FUNCTION_BLOCK FB_SimpleNciSequence
VAR_INPUT
	bExecute			: BOOL;
END_VAR
VAR_OUTPUT
	bBusy				: BOOL;
	bError				: BOOL;
	bDone				: BOOL;
END_VAR
VAR_IN_OUT
	stX					: AXIS_REF;
	stY					: AXIS_REF;
	stZ					: AXIS_REF;
	stQ1				: AXIS_REF;
	stQ2				: AXIS_REF;
	stQ3				: AXIS_REF;
	stItpToPlc			: NCTOPLC_NCICHANNEL_REF;
	stPlcToItp			: PLCTONC_NCICHANNEL_REF;
END_VAR
VAR
	nState				: UDINT	:= 0;
	nErrorState			: UDINT;
	
	fbBuildGroup		: CfgBuildExt3DGroup;
	fbLoadGCode			: ItpLoadProgEx;
	fbStartGCode		: ItpStartStopEx;
	fbClearGroup		: CfgReconfigGroup;
	fbConfirmHsk		: ItpConfirmHsk;
	
	nInterpreterState	: UDINT	:= 0;
	bConfirmHsk			: BOOL	:= FALSE;
	
//	sPrgName			: STRING(255) := 'GST_SampleFunctions.nc'; //'first.nc';
//	sPrgName			: STRING(255) := 'first.nc'; //'';
//	sPrgName			: STRING(255) := 'sample.nc'; //'';
	sPrgName			: STRING(255) := 'functionsExample.nc'; //'';
	
	
END_VAR

CASE nState OF
0:
	IF bExecute THEN
		bBusy	:= TRUE;
		bDone	:= FALSE;
		bError	:= FALSE;
		nErrorState	:= nState;
		nState	:= 10;
	END_IF	
	
10:
	// first build interpolation group 
	nInterpreterState	:= ItpGetStateInterpreter(sNciToPlc:=stItpToPlc);
	IF nInterpreterState = Tc2_NCI.NCI_INTERPRETER_IDLE THEN
		fbBuildGroup(
			bExecute	:= TRUE, 
			nGroupId	:= ItpGetGroupId(sNciToPlc:=stItpToPlc) , 
			nXAxisId	:= stX.NcToPlc.AxisId, 
			nYAxisId	:= stY.NcToPlc.AxisId, 
			nZAxisId	:= stZ.NcToPlc.AxisId, 
			nQ1AxisId	:= stQ1.NcToPlc.AxisId, 
			nQ2AxisId	:= stQ2.NcToPlc.AxisId, 
			nQ3AxisId	:= stQ3.NcToPlc.AxisId, 
			nQ4AxisId	:= 0, 
			nQ5AxisId	:= 0, 
			tTimeOut	:= , 
			bBusy		=> , 
			bErr		=> , 
			nErrId		=> );
			
		IF NOT fbBuildGroup.bBusy THEN
			IF NOT fbBuildGroup.bErr THEN
				nState	:= 20;
			ELSE
				(* add error handling *)
				nErrorState	:= nState;
				bBusy	:= FALSE;
				bError	:= TRUE;
				nState	:= 9999;
			END_IF
			fbBuildGroup(bExecute:=FALSE); 
		END_IF
	END_IF
	
20:
	// load g-code file 
	// pls. ensure that first.nc is available in TwinCAT\MC\NCI-folder 
	fbLoadGCode(
		sNciToPlc	:= stItpToPlc, 
		bExecute	:= TRUE, 
		sPrg		:= sPrgName, 
		nLength		:= INT_TO_UDINT(LEN(sPrgName)), 
		tTimeOut	:= , 
		bBusy		=> , 
		bErr		=> , 
		nErrId		=> );
		
	IF NOT fbLoadGCode.bBusy THEN
		IF NOT fbLoadGCode.bErr THEN
			nState	:= 30;
		ELSE
			(* add error handling *)
			nErrorState	:= nState;
			bBusy	:= FALSE;
			bError	:= TRUE;
			nState	:= 9999;				
		END_IF
		fbLoadGCode(sNciToPlc:=stItpToPlc, bExecute:=FALSE); 
	END_IF
	
30:
	// we have to check the status of the interpreter. It has to be in ready state, in case of loading the program successfully.
	nInterpreterState	:= ItpGetStateInterpreter(sNciToPlc:=stItpToPlc);
	IF nInterpreterState = Tc2_NCI.NCI_INTERPRETER_READY THEN
		nState	:= 40;
	ELSE
		(* add error handling *)
		nErrorState	:= nState;
		bBusy	:= FALSE;
		bError	:= TRUE;
		nState	:= 9999;				
	END_IF
	
40:
	// start g-code file
	fbStartGCode(
		bStart		:=TRUE, 
		bStop		:=FALSE, 
		tTimeOut	:= , 
		sNciToPlc	:= stItpToPlc, 
		bBusy		=> , 
		bErr		=> , 
		nErrId		=> );
		
	IF NOT fbStartGCode.bBusy THEN
		IF NOT fbStartGCode.bErr THEN
			nState	:= 50;
		ELSE	
			(* add error handling *)
			nErrorState	:= nState;
			bBusy	:= FALSE;
			bError	:= TRUE;
			nState	:= 9999;				
		END_IF
		fbStartGCode( bStart:=FALSE, sNciToPlc:= stItpToPlc ); 
	END_IF
	
50:
	// check state, again - we are at least not in ready state for several ticks
	// this is to ensure that we don't indicate program has finished, before we have started 
	nInterpreterState	:= ItpGetStateInterpreter(sNciToPlc:=stItpToPlc);
	IF nInterpreterState <> Tc2_NCI.NCI_INTERPRETER_READY THEN
		// nci is running
		nState	:= 60;
	END_IF

60:
	nInterpreterState	:= ItpGetStateInterpreter(sNciToPlc:=stItpToPlc);
	IF	nInterpreterState = Tc2_NCI.NCI_INTERPRETER_READY THEN
		// program has finished
		nState	:= 70;
	ELSIF nInterpreterState = Tc2_NCI.NCI_INTERPRETER_ABORTED THEN
		// a run-time error occured - this could be a lag error or something else... 
		// add error handling
		;
	END_IF	
	
70:
	// program has finished 
	// now clear interpolation group 
	fbClearGroup(
		bExecute	:= TRUE, 
		nGroupId	:= ItpGetGroupId(sNciToPlc:=stItpToPlc) , 
		tTimeOut	:= , 
		bBusy		=> , 
		bErr		=> , 
		nErrId		=> );
		
	IF NOT fbClearGroup.bBusy THEN
		IF NOT fbClearGroup.bErr THEN
			nState	:= 80;
		ELSE
			(* add error handling *)
			nErrorState	:= nState;
			bBusy	:= FALSE;
			bError	:= TRUE;
			nState	:= 9999;				
		END_IF
		fbClearGroup(bExecute:=FALSE); 
	END_IF
80:
	bDone	:= TRUE;
	bBusy	:= FALSE;
	IF NOT bExecute THEN
		nState	:= 0;
	END_IF
	
9999:
	// error state 
	IF NOT bExecute THEN
		nState	:= 0;
		bError	:= FALSE;
	END_IF
END_CASE

// handling of m-functions is done outside statemachine
// all m-functions are directly confiremd. In a real application we have of course to consider the m-function numbers to turn on/off certain functions in the machine.
IF ItpIsHskMFunc(stItpToPlc) AND NOT fbConfirmHsk.bBusy THEN
	bConfirmHsk	:= TRUE;
ELSE	
	bConfirmHsk	:= FALSE;
END_IF	

fbConfirmHsk(
	bExecute:=bConfirmHsk , 
	sNciToPlc:=stItpToPlc , 
	sPlcToNci:=stPlcToItp , 
	bBusy=> , 
	bErr=> , 
	nErrId=> );

END_FUNCTION_BLOCK

(* stored: Version 1.1.0.1, ProductVersion 3.1.4024.10
   POU FB_SimpleNciSequence: Id {4f24b964-7729-4762-90ad-698d0a17343d}, SpecialFunc None *)
